(* PLC project CHL-DZ-BJDX-11 宁波数字孪生（东方理工）研究院制备薄层色谱全自动化工作站.project, Inovance company InoProShop(V1.9.1.6) InoProShop(V1.9.1.6) *)
(* stored: creationDateTime 2026-06-18T00:43:55.0933428, modificationDateTime 2026-06-17T21:37:38.1461871 *)

ACTION A20_collect_收集:
            ton[1](IN:=收集step=10,PT:=T#0.5S);
ton[2](IN:=收集step=30,PT:=T#10S);
R_TRIG[5](CLK:=%MX2005.5 , Q=> );  //泵空闲中
CASE 收集step OF
	0 :
		IF collect_forward_instructions<>'' THEN
			收集进液自动:=TRUE;
			
			
		END_IF
		IF %MW1300=0 AND 泵站位符=FALSE  THEN
			转发转存:=collect_forward_instructions; 
			%MW1300:=LEN(STR:= 转发转存);   //发送字节数
			泵站位符:=TRUE;
			收集step:=10;
		END_IF
	10:
		IF %MW1300=0 AND ton[1].Q THEN
			转发转存:='/3Q$R';          //查询泵状态指令
			%MW1300:=LEN(STR:= 转发转存);
		END_IF
		
		
		IF R_TRIG[5].Q THEN
			泵站位符:=FALSE;
			收集step:=20;
		END_IF
	

	20:
		IF TRUE  THEN    //注射泵完成//
			转发转存:='';
			%MW300:=128;
			收集进液自动:=FALSE;
			收集排液自动:=TRUE;
			收集正压排液自动:=TRUE;
			收集计数:=收集计数+1;
			收集step:=30;
		END_IF
	30:
		IF ton[2].Q THEN
			TON_0(IN:=TRUE, PT:=T#5S , Q=> , ET=> );
			IF 收集计数>=collect_count AND TON_0.Q THEN
				收集计数:=0;
				收集step:=40;
			ELSE
				收集排液自动:=FALSE;
				收集正压排液自动:=FALSE;
				收集step:=0;
			END_IF
		END_IF
	40:
		
			收集排液自动:=FALSE;
			收集正压排液自动:=FALSE;
			collect_OK:=TRUE;
			收集step:=0;

		

		
END_CASE
          
END_ACTION

ACTION A00_initialization_初始化:
            R_TRIG[1](CLK:=%MX2005.5 , Q=> );  //泵空闲中

//初始化流程
CASE 初始化STEP OF
	0:
		收集下压气缸手动:=FALSE;
		收集下压气缸自动:=FALSE;
		收集夹持气缸手动:=FALSE;
		收集夹持气缸自动:=FALSE;
		收集升降气缸手动:=FALSE;
		收集升降气缸自动:=FALSE;
		收集伸缩气缸手动:=FALSE;
		收集伸缩气缸自动:=FALSE;
		收集进液手动:=FALSE;
		收集进液自动:=FALSE;
		收集排液手动:=FALSE;
		收集排液自动:=FALSE;
		收集正压排液手动:=FALSE;
		收集正压排液自动:=FALSE;
		溶液收集瓶定位手动:=FALSE;
		收集工位允许放收集瓶:=FALSE;
		收集工位允许放收集器:=FALSE;
		收集工位允许机器人退出工位:=FALSE;
		收集工位允许机器人取收集瓶放暂存工位:=FALSE;
		收集工位允许取收集器:=FALSE;
		收集工位机器人取收集器放回暂存工位:=FALSE;
		
	
		收集工位放收集瓶完成:=FALSE;
		收集工位放收集器到工位:=FALSE;
	
		收集工位机器人退出完成:=FALSE;
		
		收集工位机器人放收集瓶到暂存工位完成:=FALSE;
		
		收集工位机器人到达收集器位置:=FALSE;

		collect_prepare_OK:=FALSE;
		collect_OK:=FALSE;
		收集工位放收集器完成:=FALSE;
		收集step:=0;
		准备step:=0;
		搬运step:=0;
		IF %MW1300=0 AND NOT 泵站位符 THEN
			泵站位符:=TRUE;
			转发转存:='/3Z0,2,2R$R';     //泵初始化指令 
			%MW1300:=LEN(STR:= 转发转存);   //发送字节数
			初始化STEP:=10;
		END_IF
	10:
		IF %MW1300=0 THEN
			转发转存:='/3Q$R';          //查询泵状态指令
			%MW1300:=LEN(STR:= 转发转存);
		END_IF
		
		IF R_TRIG[1].Q THEN
			泵站位符:=FALSE;
			泵初始化完成:=TRUE;
			初始化STEP:=0;
		END_IF
END_CASE
	
	
	
	
	
	
	
	
	
	

		


          
END_ACTION

ACTION A30_transport_物料搬运:
            

CASE 搬运step OF
	0 :                     //复位气缸
		收集下压气缸自动:=FALSE;
		
		搬运step:=5;
	5:
		IF 收集平台下压气缸原点 THEN
			收集升降气缸自动:=FALSE;
			搬运step:=10;
		END_IF
	10:                    //复位伸缩气缸
		IF 收集平台升降气缸原点 THEN
			收集伸缩气缸自动:=TRUE;
			搬运step:=20;
		END_IF
	20:                    //允许机器人收集瓶
		IF 收集平台推出气缸动点 THEN
			收集工位允许机器人取收集瓶放暂存工位:=TRUE;
			搬运step:=30;
		END_IF
	30:
		IF 收集工位机器人放收集瓶到暂存工位完成 THEN
			收集工位允许机器人取收集瓶放暂存工位:=FALSE;
			收集工位机器人放收集瓶到暂存工位完成:=FALSE;
			收集伸缩气缸自动:=FALSE;
			收集工位允许取收集器:=TRUE;
			搬运step:=40;
		END_IF
	40:
		IF 收集工位机器人到达收集器位置 THEN
				收集工位机器人到达收集器位置:=FALSE;
			收集夹持气缸自动:=FALSE;
			收集工位允许取收集器:=FALSE;
			搬运step:=50;
		END_IF
	50:
		IF 收集平台夹持气缸原点 THEN
			收集工位机器人取收集器放回暂存工位:=TRUE;
			搬运step:=60;
		END_IF
	60:
		 IF 收集工位放收集器完成 THEN
		 	搬运step:=0;
		 END_IF
		
		
		

END_CASE
          
END_ACTION

ACTION A10_preparation_准备:
            //准备工作
CASE 准备step OF	
	0:
		IF 收集平台夹持气缸原点 AND 收集平台下压气缸原点 THEN
		收集工位允许放收集器:=TRUE;
		准备step:=10;
		END_IF
	10:
		IF 收集工位放收集器到工位 THEN
			收集夹持气缸自动:=TRUE;
			收集工位允许放收集器:=FALSE;
			准备step:=20;
		END_IF
	20:
		IF 收集平台夹持气缸动点 THEN
			收集工位允许机器人退出工位:=TRUE;
			准备step:=30;
		END_IF
		
	30:
		IF 收集工位机器人退出完成 THEN
			
			收集工位机器人退出完成:=FALSE;
			收集工位允许机器人退出工位:=FALSE;
			准备step:=40;
		END_IF
	40 :
		IF 收集平台推出气缸原点 AND NOT 收集平台瓶子有无传感器 THEN
			收集伸缩气缸自动:=TRUE;
			准备step:=50;
		END_IF
	50:
		IF 收集平台推出气缸动点 THEN
			收集工位允许放收集瓶:=TRUE;
			准备step:=60;
		END_IF
	60:
	    IF 收集工位放收集瓶完成 THEN
	    	收集工位允许放收集瓶:=FALSE;
			收集工位放收集瓶完成:=FALSE;
			收集伸缩气缸自动:=FALSE;
			准备step:=70;
	    END_IF
	70:
		IF 收集平台推出气缸原点 AND 收集平台瓶子有无传感器 THEN
			收集升降气缸自动:=TRUE;
			准备step:=80;
		ELSIF 收集平台推出气缸原点 AND NOT 收集平台瓶子有无传感器 THEN
			收集伸缩气缸自动:=FALSE;
			准备step:=40;
		END_IF

	80:
		IF 收集平台升降气缸动点  THEN
			收集下压气缸自动:=TRUE;
			collect_prepare_OK:=TRUE;
			准备step:=0;
		END_IF
		
END_CASE
          
END_ACTION

PROGRAM Collection_process_收集流程
  VAR
    准备step : INT;
    收集step : INT;
    TON_0 : TON;
    搬运step : INT;
    ton3s : TON;
    ton5s : TON;
    i : INT;
    stepTimer : TON;
    R_TRIG : ARRAY[1..5] OF R_TRIG;
    泵初始化完成 : BOOL;
    初始化STEP : INT;
    ton : ARRAY[1..10] OF TON;
  END_VAR

            // TON自复位：Q变TRUE后IN立即变FALSE，下周期复位，形成循环脉冲
ton3s(IN := bEnable AND NOT ton3s.Q, PT := T#3S);

// Q脉冲时翻转输出（Q仅维持一个周期，无需上升沿检测）
IF ton3s.Q THEN
    bOutput := NOT bOutput;
END_IF

// ── 1. 急停联锁（最高优先级）──
IF NOT 急停 THEN
    collect_Step  := 0;
    collect_Done  := FALSE;
    collect_Error := TRUE;
    collect_Busy  := FALSE;
	准备step:=0;
	收集step:=0;
	搬运step:=0;
	初始化STEP:=0;
	泵初始化完成:=FALSE;
    stepTimer(IN := FALSE, PT := T#0S);
    RETURN;
END_IF

// ── 2. 复位脉冲（用于错误恢复 / 强制清状态）──
IF collect_Reset THEN
    collect_Step  := 0;
    collect_Done  := FALSE;
    collect_Error := FALSE;
    collect_Busy  := FALSE;
    stepTimer(IN := FALSE, PT := T#0S);
    RETURN;
END_IF

// ── 3. Enable=FALSE 时清 Done（次周期复位握手）──
//    上位机收到 Done 后会拉低 collect_Enable，本段确保下一周期 Done 自动归零，
//    避免 Done 残留导致 step 0 误判。
IF NOT collect_Enable THEN
    collect_Done := FALSE;
END_IF

// ── 4. 派生 collect_Busy（写者唯一：本 POU 是唯一写者，禁止他处赋值）──
collect_Busy := (collect_Step >= 10)
                    AND (collect_Step <= 80)
                    AND (NOT collect_Done);






IF MODE_State=1 THEN
	CASE collect_Step OF
		0 :                      // 空闲：等待 Enable 上升
			 IF collect_Enable AND (NOT collect_Done) THEN
				collect_Step := 5;
			 END_IF
		
		5:	
		    A00_initialization_初始化();
			IF 收集平台下压气缸原点 AND 收集平台夹持气缸原点 AND 收集平台升降气缸原点 AND 收集平台推出气缸原点 AND 泵初始化完成 THEN
				collect_Step:=10;
				泵初始化完成:=FALSE;
			END_IF
			
			
				
		10:                    //就位
				A10_preparation_准备();
			IF collect_prepare_OK THEN
				collect_prepare_OK:=FALSE;
				collect_Step:=20;
			END_IF
			
			
			
		20:                    //收集    	
			A20_collect_收集();
			IF collect_OK THEN
				
				FOR i := 1 TO collect_count BY 1 DO
					;   // 占位：单次打液动作（实机替换为真实调用）
				END_FOR
				collect_OK:=FALSE;
				collect_Step:=30;
			END_IF
			
			
		30:                    //物料搬运
			A30_transport_物料搬运();
			 IF 收集工位放收集器完成 THEN
				 收集工位放收集器完成:=FALSE;
				collect_Done := TRUE;
				collect_Step:=0;
			 END_IF	
			 
			 
		90: // 故障：等待外部 collect_Reset 脉冲（已在顶部统一处理）
			collect_Error := TRUE;   // 故障态本身不动作，仅等待复位
	END_CASE
END_IF











































































































          
END_PROGRAM
